FUNCTION_BLOCK FB_ArgStack
VAR_INPUT
END_VAR
VAR_OUTPUT
END_VAR
VAR
	pStackMemory			: POINTER TO BYTE;
	nStackMemorySize		: DINT;
	nCurrOfsetInStack		: DINT;
END_VAR
VAR CONSTANT
	ARG_HEADER_SIZE			: DINT := 2;
END_VAR

PROPERTY PROTECTED ArgDataAvailableSize : DINT
GET
ArgDataAvailableSize := MAX(0, RemainingMemorySize - ARG_HEADER_SIZE);
END_GET
END_PROPERTY

PROPERTY PROTECTED ArgDataOffset : DINT
GET
ArgDataOffset := nCurrOfsetInStack + ARG_HEADER_SIZE;
END_GET
END_PROPERTY

PROPERTY PUBLIC ArgDataPointer : POINTER TO BYTE
GET
ArgDataPointer := ADR(pStackMemory[ArgDataOffset]);
END_GET
END_PROPERTY

PROPERTY PROTECTED ArgSize : BYTE
GET
ArgSize := pStackMemory[nCurrOfsetInStack + 1];
END_GET
SET
pStackMemory[nCurrOfsetInStack + 1] := ArgSize;
END_SET
END_PROPERTY

PROPERTY PROTECTED ArgType : BYTE
GET
ArgType := pStackMemory[nCurrOfsetInStack];
END_GET
SET
pStackMemory[nCurrOfsetInStack] := ArgType;
END_SET
END_PROPERTY

PROPERTY PROTECTED AtEndOfMemory : BOOL
GET
AtEndOfMemory := RemainingMemorySize < ARG_HEADER_SIZE;
END_GET
END_PROPERTY

METHOD PUBLIC Clear
nCurrOfsetInStack := 0;

IF nStackMemorySize > 0 THEN
	// Zero stack memory
	F_MemSet(
		pDestAddr:= pStackMemory,
		nWithChar:= 0,
		stDestSize:= DINT_TO_SIZE(nStackMemorySize));
END_IF
END_METHOD

METHOD FB_init : BOOL
VAR_INPUT
	bInitRetains		: BOOL; // if TRUE, the retain variables are initialized (warm start / cold start)
	bInCopyCode			: BOOL;  // if TRUE, the instance afterwards gets moved into the copy code (online change)
	pStackMemory		: POINTER TO BYTE;
	nStackMemorySize	: DINT;
END_VAR
SetMemory(pStackMemory, nStackMemorySize);
END_METHOD

PROPERTY PUBLIC MemoryPointer : POINTER TO BYTE
GET
MemoryPointer := pStackMemory;
END_GET
END_PROPERTY

PROPERTY PUBLIC MemorySize : DINT
GET
MemorySize := nStackMemorySize;
END_GET
END_PROPERTY

PROPERTY PROTECTED RemainingMemorySize : DINT
GET
RemainingMemorySize := nStackMemorySize - nCurrOfsetInStack;
END_GET
END_PROPERTY

METHOD PUBLIC SetMemory
VAR_INPUT
	pStackMemory		: POINTER TO BYTE;
	nStackMemorySize	: DINT;
END_VAR
THIS^.pStackMemory := pStackMemory;

IF THIS^.pStackMemory <> 0 THEN
	THIS^.nStackMemorySize := nStackMemorySize;
ELSE
	THIS^.nStackMemorySize := 0;
END_IF

THIS^.nCurrOfsetInStack := 0;
END_METHOD

PROPERTY PUBLIC UsedMemorySize : DINT
GET
UsedMemorySize := nCurrOfsetInStack;
END_GET
END_PROPERTY

END_FUNCTION_BLOCK

(* stored: Version 1.1.0.1, ProductVersion 3.1.4024.15
   POU FB_ArgStack: Id {5aca428e-fddd-4368-a23a-daa0a6193ea2}, SpecialFunc None
   Property ArgDataAvailableSize: Id {de7a8127-1eb8-47f6-ba84-c0222375861f}
   Get Get: Id {62763f37-3a46-49f7-bd23-261f0b6844d2}
   Property ArgDataOffset: Id {5b091e0b-9606-4c96-ad76-a9ddea1d6a54}
   Get Get: Id {ed618d43-6339-4f85-a02b-661e5cae8e5c}
   Property ArgDataPointer: Id {67e77f93-0c7c-464e-a41e-e717e057f691}
   Get Get: Id {306a822d-c915-4f35-9e83-9df596cd217d}
   Property ArgSize: Id {2f9ac1b1-db36-4120-b5d3-f4ba1c0bc294}
   Get Get: Id {465a96fe-684b-40e5-9788-5d17b2732bc4}
   Set Set: Id {83a45f2e-62dd-49c4-89cd-72526e7a852d}
   Property ArgType: Id {8dff9f69-cd50-4b55-b47c-4d2c0dbd81f3}
   Get Get: Id {b6bbd970-8717-45a9-ac72-4b5bb9ae30a3}
   Set Set: Id {acd10166-0626-4379-b470-da6d3d22000a}
   Property AtEndOfMemory: Id {94135612-bd36-4768-86c4-dc4015449b57}
   Get Get: Id {8a3cea2c-ae6b-4de9-9a19-eba2af230cfd}
   Method Clear: Id {61ae53d5-0357-48cb-807c-17cbeada3a8c}
   Method FB_init: Id {b1481970-1f76-489f-910d-b0f425ca9ae4}
   Property MemoryPointer: Id {580d5b7a-81bd-464b-a9c8-40858491b0de}
   Get Get: Id {3b929468-ca7f-4b3c-83fe-f333e6202ca2}
   Property MemorySize: Id {ad6e4f2c-14b1-439f-87bf-3767e39cb9d5}
   Get Get: Id {7c136861-7956-4188-adf4-1403b21a7a06}
   Property RemainingMemorySize: Id {ee0f045c-05eb-433a-a6ee-b87169491f95}
   Get Get: Id {b7097647-0e9f-456a-a402-875ec97504a9}
   Method SetMemory: Id {eb4dabce-185b-4416-838b-fe62834036b5}
   Property UsedMemorySize: Id {ef9444e9-bd18-4f67-a51a-a3d21b0e8701}
   Get Get: Id {a01f0c64-3e54-476f-ae01-3645e39de6cd} *)
